FUNCTION_BLOCK FB_Semaforo
VAR_INPUT
	bON			:BOOL;
	sColore		:int;
	bBlink		:BOOL;
END_VAR
VAR_OUTPUT
	semaforo	:ES_SEMAFORO;
END_VAR
VAR
	_tmrBlink	:ton;
	_bAccesa	:BOOL;
END_VAR


//1: BLU
//2: VERDE
//4: ROSSO
//6: ARANCIO

semaforo.analog0:= 0;
semaforo.analog1:= 0;
semaforo.analog2:= 0;
semaforo.analog3:= 0;
semaforo.analog4:= 0;
semaforo.analog5:= 0;
		
IF bBlink THEN
	_tmrBlink(IN:= bON, PT:=T#1000MS);
	IF _tmrBlink.Q THEN
		_tmrBlink(IN:= FALSE);
		_bAccesa:= NOT _bAccesa;
	END_IF
ELSE
	_bAccesa:=TRUE;
END_IF
		
IF bON THEN

	CASE sColore OF
				
	1: //BLU:
		IF _bAccesa THEN
			semaforo.analog1:= 1;
		END_IF 
		
	2: //ROSSO:
		IF _bAccesa THEN
			semaforo.analog2:= 4;
		END_IF
		
	3: //VERDE:
		IF _bAccesa THEN
			semaforo.analog3:= 2;
		END_IF
		
	4: //ARANCIO:
		IF _bAccesa THEN
			semaforo.analog4:= 6;
		END_IF
				
	
	END_CASE


END_IF

END_FUNCTION_BLOCK

(* stored: Version 1.1.0.1, ProductVersion 3.1.4022.12
   POU FB_Semaforo: Id {29b95473-734d-4818-9fec-b31c8f88d9dd}, SpecialFunc None *)
